{attribute 'qualified_only'}
{attribute 'strict'}
TYPE E_ReferenceCommand : (None, Home, Start, Stop, Abort, Reset); END_TYPE

(* stored: Version 1.1.0.1
   DUT E_ReferenceCommand: Id {00c1196b-aa56-41b8-ab7d-c1b7bf644f85} *)
